{attribute 'qualified_only'}
{attribute 'strict'}
{attribute 'to_string'}
{attribute  'hide'}
TYPE E_EventType :
(
	Info:=0,
	Warning:=1,
	Error:=2
);
END_TYPE

(* stored: Version 1.1.0.1, ProductVersion 3.1.4024.6
   EnumerationTextList E_EventType: Id {d829e07a-e525-4d07-a9ea-97334815ebee} *)
